// TwinCAT 3 PLC project RealFFT
// ProgramVersion: 3.1.4020.10
// libraries:
//   Tc2_Standard, * (Beckhoff Automation GmbH)
//   Tc2_System, * (Beckhoff Automation GmbH)
//   Tc2_Utilities, * (Beckhoff Automation GmbH)
//   Tc3_CM, * (Beckhoff Automation GmbH)
//   Tc3_CM_Base, * (Beckhoff Automation GmbH)
//   Tc3_Module, * (Beckhoff Automation GmbH)
//   Tc3_MultiArray, * (Beckhoff Automation GmbH)
// project tree:
//   DUTs/Error Monitoring/ ST_HRErrHist.TcDUT
//   DUTs/ E_AnalysisIDs.TcDUT
//   DUTs/Function Generator/ E_FunctionType.TcDUT
//   GVLs/ GVL_Constants.TcGVL
//   / PlcTask.TcTTO, PlcTaskCM.TcTTO
//   POUs/Error Monitoring/ FB_HRErrHist.TcPOU
//   POUs/Function Generator/ FB_FunctionGenerator.TcPOU
//   POUs/ MAIN.TcPOU, MAIN_CM.TcPOU
// real-time tasks:
//   TASK PlcTaskCM: cycle T#5ms, priority 6, ADS port 350
//   TASK PlcTask: cycle T#1ms, priority 4, ADS port 351

CONFIGURATION RealFFT
    RESOURCE PLC ON TwinCAT3
        TASK PlcTask(INTERVAL := T#1ms, PRIORITY := 4);
        TASK PlcTaskCM(INTERVAL := T#5ms, PRIORITY := 6);
        PROGRAM MAIN WITH PlcTask : MAIN;
        PROGRAM MAIN_CM WITH PlcTaskCM : MAIN_CM;
    END_RESOURCE
END_CONFIGURATION

// ---- DUTs/Error Monitoring/ST_HRErrHist.TcDUT
TYPE ST_HRErrHist :
STRUCT
{attribute 'displaymode':='hex'}
	hrErrCode	: HRESULT;
	sErrSource	: STRING(63);
	nErrCount	: UDINT;
END_STRUCT
END_TYPE

// ---- DUTs/E_AnalysisIDs.TcDUT
TYPE E_AnalysisIDs :
(
	(* analysis chain *)
	eID_Source := 1,
	eID_FFT,
	eID_Sink
	
) UDINT;
END_TYPE

// ---- DUTs/Function Generator/E_FunctionType.TcDUT
{attribute 'qualified_only'}
TYPE E_FunctionType :
(
	Sine,		// typical for vibrations originating from rotating machine
	Square,		// mixed sine signals good for analyzing spectrum
	Pulse,		// mixed sine signals good for analyzing spectrum
	Triangular,	// mixed sine signals good for analyzing spectrum
	Sawtooth,	// ramp-type vibrations, continuously increasing
	AM			// amplitude modulation: typical for vibrations originating from gear-tooth failure or bearing faults
);
END_TYPE

// ---- GVLs/GVL_Constants.TcGVL
VAR_GLOBAL CONSTANT
	
	cOversamples 	: UDINT 	:= 10;				 // number of oversamples
	cFFTLength		: UDINT		:= 2048;			 // length of FFT 
	cBufferLength	: UDINT		:= cFFTLength;	     // attention: needs to be equal to cFFTLength (no overlap)	
	cFFTResult 		: UDINT 	:= cFFTLength/2+1;	 // result of mag. spectrum - cFFTLength/2+1
		
END_VAR

// ---- POUs/MAIN.TcPOU
PROGRAM MAIN

VAR CONSTANT
    cInitSource			: ST_MA_MultiArray_InitPars 
							:= ( eTypeCode := eMA_TypeCode_LREAL, nDims := 1, aDimSizes := [cBufferLength]);	
END_VAR

VAR
	(* Input *)
	nInputSelection		: UDINT := 1;						// Switch between hardware and function generator	
	nSample				: UDINT;                            
	aEl3632 AT %I*		: ARRAY[1..cOversamples] OF INT;	// Input from hardware e.g. EL3632
	
	(* Signal Generator *)
	fbFunctionGenerator	: FB_FunctionGenerator;
	fSetFrequency		: LREAL := 200;		// Hz
	fSetAmplitude		: LREAL := 13;		// peak amplitude of sin signal, in Volts		
    fDC					: LREAL := 7;       // Amplitude of DC	
	
	(* Source buffers *)	
	aBuffer				: ARRAY[1..cOversamples] OF LREAL;				// local varibale -> to source				
	fbSource			: FB_CMA_Source :=(	stInitPars := cInitSource, 
											nOwnID := eID_Source, 
											aDestIDs := [eID_FFT]);		// Initialize source buffers
	(* Result buffers *)										
	aSpectrumResult		: ARRAY[1..cFFTResult] OF LCOMPLEX;				// local result variable <- from sink
    fbSink				: FB_CMA_Sink := (nOwnID := eID_Sink);			// Initialize sink buffers
	
	
	(* post-processing of fft *)
	nCountResults		: ULINT;							// increments for every fft calculation
	bCalculate			: BOOL;								// true if fft calculation ready	
	SpectrumAbs         : ARRAY[1..cFFTResult] OF LREAL; 	// magnitude spectrum variable 
	(* max amplitude calculation *)
	fMaxAmpl			: LREAL;
	nIdxOfMaxAmpl		: UDINT;							// index of max amplitude in spectrum result array 
	(* frequency calculation *)
	fSampleTaskCycleTime: LREAL := 1; // ms
	fSampleRate			: LREAL;      // Hz  ( sample rate = oversampling factor / cycle time )
	fResolution			: LREAL;      // Hz/Idx
	fFrequency			: LREAL;      // Hz	
	
	(* error monitoring *)
	fbErrHist			: FB_HRErrHist;

END_VAR

(* Input *) 
CASE nInputSelection OF
	0:  (* input from EL3632 *)
		FOR nSample := 1 TO cOversamples DO
			aBuffer[nSample] := INT_TO_LREAL(aEl3632[nSample]);
		END_FOR
	1:  (* signal generator *)		
		fbFunctionGenerator(	fFrequency 	:= fSetFrequency,
								fAmplitude 	:= fSetAmplitude,
								eFunction 	:= E_FunctionType.Sine,
								aSignal		:= aBuffer );		
        // add DC to signal
		FOR nSample := 1 TO cOversamples DO
			aBuffer[nSample] := fDC+aBuffer[nSample];
		END_FOR								
END_CASE					

(* Call source to collect data *)
fbSource.Input1D( pDataIn 			:= ADR(aBuffer),
				  nDataInSize 		:= SIZEOF(aBuffer), 
				  eElementType 		:= eMA_TypeCode_LREAL,
				  nWorkDim 			:= 0,
				  pStartIndex		:= 0,
				  nOptionPars		:= cCMA_Option_MarkInterruption ); 
IF fbSource.bError THEN
	fbErrHist.AddError(bErr:=TRUE, hrErrCode:=fbSource.hrErrorCode, sErrSource:='MAIN.fbSource'); // error monitoring
	// ToDo: if error
END_IF


(* Push results to sink *)
fbSink.Output1D(	pDataOut 		:= ADR(aSpectrumResult), 
					nDataOutSize 	:= SIZEOF(aSpectrumResult), 
					eElementType 	:= eMA_TypeCode_LCOMPLEX, 
					nWorkDim 		:= 0,
					nElements		:= 0,
					pStartIndex 	:= 0,
					nOptionPars		:= 0,
					bNewResult		=> bCalculate );
IF fbSink.bError THEN
	fbErrHist.AddError(bErr:=TRUE, hrErrCode:=fbSink.hrErrorCode, sErrSource:='MAIN.fbSink'); // error monitoring
	// ToDo: if error
END_IF

(* post-process fft result *)
IF bCalculate THEN
	nCountResults := fbSink.nCntResults;
	
	// Calculate absolute value as aSpectrumResult is of complex type
	FOR nSample := 1 TO cFFTResult DO			   	   
	   SpectrumAbs[nSample] := SQRT(aSpectrumResult[nSample].re * aSpectrumResult[nSample].re + aSpectrumResult[nSample].im * aSpectrumResult[nSample].im);
       
	   // scale spectrum
	   IF nSample = 1 THEN
		   SpectrumAbs[nSample] := SpectrumAbs[nSample]/cFFTLength;   // scale DC value
	   ELSE
		   SpectrumAbs[nSample] := 2*SpectrumAbs[nSample]/cFFTLength; // scale frequencies not equal to 0
	   END_IF
	   
	   
	END_FOR;
	
	IF NOT lrealisnan(SpectrumAbs[1]) THEN
		// Calculate max amplitude in spectrum
		fMaxAmpl := 0;
		FOR nSample:=1 TO cFFTResult DO
			IF SpectrumAbs[nSample] > fMaxAmpl THEN
				fMaxAmpl := SpectrumAbs[nSample];
				nIdxOfMaxAmpl := nSample;
			END_IF
		END_FOR
		
		// Calculate frequency for max amplitude [ frequency = index * (sample rate / FFT length) ]
		fSampleRate := cOversamples * (1000.0 / fSampleTaskCycleTime);
		fResolution := fSampleRate / cFFTLength;
		fFrequency := (nIdxOfMaxAmpl-1) * fResolution;	 // -1 to consider DC = 0*fResolution
	END_IF

	
END_IF

END_PROGRAM

// ---- POUs/Function Generator/FB_FunctionGenerator.TcPOU
// generates a signal build up by the specified function type. v1.6
FUNCTION_BLOCK FB_FunctionGenerator
VAR_INPUT
	bEnable		: BOOL 	:= TRUE;	// set TRUE to generate the specified signal; set FALSE to reset the signal buffer
	fFrequency	: LREAL := 1000;	// in [Hz]
	fAmplitude	: LREAL := 1;
	fOffset		: LREAL	:= 0;	
	nDutyCycle	: UINT 	:= 50;		// in [%] (for pulse function)
	eFunction	: E_FunctionType := E_FunctionType.Sine;	
END_VAR
VAR_IN_OUT
	aSignal		: ARRAY[1..cOversamples] OF LREAL;
END_VAR
VAR_OUTPUT
	bError		: BOOL;
END_VAR

VAR
	bInit						: BOOL := TRUE;
	fbGetTaskIdx				: GETCURTASKINDEX;
	
	fLastFrequency				: LREAL;		// in [Hz]
	fLastAmplitude				: LREAL;
	fLastOffset					: LREAL;
	nLastDutyCycle				: UINT;
	eLastFunction				: E_FunctionType;
	
	nSamples					: UDINT;
	fCycleTime					: LREAL;		// in [s]
	fDelta						: LREAL;		// amplitude delta per sample
	fPhase						: LREAL;		// in [°]
	nSign						: INT := 1;		// 1 or -1
	fLastSignalValue			: LREAL;		// amplitude
	fPeriod						: LREAL;		// in [s]
	fAngularIncrement			: LREAL;		// in [°]
	fAngularIncrementPerCycle	: LREAL;		// in [°]
	fAngularIncrementPerSample	: LREAL;		// in [°]
	(* for modulated signal (carrier signal without offset) *)
	fCarrierFrequency					: LREAL := 500;	// in [Hz] (sine)
	fCarrierAmplitude					: LREAL := 1;
	fCarrierPeriod						: LREAL;		// in [s]
	fCarrierAngularIncrement			: LREAL;		// in [°]
	fCarrierAngularIncrementPerCycle	: LREAL;		// in [°]
	fCarrierAngularIncrementPerSample	: LREAL;		// in [°]
				
END_VAR

IF bEnable THEN
	IF fLastFrequency <> fFrequency THEN
		bInit := TRUE; // For automatic initializing
		fLastFrequency := fFrequency;
	END_IF
	IF fLastAmplitude <> fAmplitude THEN
		bInit := TRUE; // For automatic initializing
		fLastAmplitude := fAmplitude;
	END_IF
	IF fLastOffset <> fOffset THEN
		bInit := TRUE; // For automatic initializing
		fLastOffset := fOffset;
	END_IF
	IF nLastDutyCycle <> nDutyCycle THEN
		bInit := TRUE; // For automatic initializing
		nLastDutyCycle := nDutyCycle;
	END_IF
	IF eLastFunction <> eFunction THEN
		bInit := TRUE; // For automatic initializing
		eLastFunction := eFunction;
	END_IF
	IF bInit THEN
		// Get task info	
		fbGetTaskIdx();
		fCycleTime := UDINT_TO_LREAL(TwinCAT_SystemInfoVarList._TaskInfo[fbGetTaskIdx.index].CycleTime) (*100ns*) / (10.0 * 1000.0 * 1000.0);	
		fLastSignalValue := 0;
		nSign := 1;
		fAngularIncrement := 0;
		// Flush out old data
		MEMSET(ADR(aSignal), 0, SIZEOF(aSignal));
		IF fFrequency > 0 AND fCycleTime > 0 THEN		
			// Calculate period, increments per plc cycle, increment per oversample
			IF cOversamples > 0 THEN			
				IF eFunction = E_FunctionType.Sine THEN
					fPeriod := 1/fFrequency;
					fAngularIncrementPerCycle := 360*(fCycleTime/fPeriod);
					fAngularIncrementPerSample := fAngularIncrementPerCycle/cOversamples;
					// no phase adjustment
					bInit := FALSE;	
				ELSIF eFunction = E_FunctionType.Square	THEN
					fPeriod := 1/fFrequency;
					fAngularIncrementPerCycle  := 360*(fCycleTime/fPeriod);
					fAngularIncrementPerSample := fAngularIncrementPerCycle/cOversamples;
					fPhase := 0.5*360;
					bInit := FALSE;
				ELSIF eFunction = E_FunctionType.Pulse THEN
					fPeriod := 1/fFrequency;
					fAngularIncrementPerCycle  := 360*(fCycleTime/fPeriod);
					fAngularIncrementPerSample := fAngularIncrementPerCycle/cOversamples;
					IF nDutyCycle > 100 THEN
						nDutyCycle := 100;
					END_IF
					fPhase := (UDINT_TO_LREAL(nDutyCycle)/100)*360;
					bInit := FALSE;					
				ELSIF eFunction = E_FunctionType.Triangular THEN
					fPeriod := 1/fFrequency;				
					fAngularIncrementPerCycle  := 360*(fCycleTime/fPeriod);
					fAngularIncrementPerSample := fAngularIncrementPerCycle/cOversamples;
					fPhase := 0.5*360; 
					fDelta := 4*(fAmplitude/(360/fAngularIncrementPerSample));				
					bInit := FALSE;
				ELSIF eFunction = E_FunctionType.Sawtooth THEN
					fPeriod := 1/fFrequency;			
					fAngularIncrementPerCycle  := 360*(fCycleTime/fPeriod);		
					fAngularIncrementPerSample := fAngularIncrementPerCycle/cOversamples;
					fDelta := fAmplitude/(360/fAngularIncrementPerSample);
					bInit := FALSE;
				ELSIF eFunction = E_FunctionType.AM THEN
					fPeriod := 1/fFrequency;
					fAngularIncrementPerCycle := 360*(fCycleTime/fPeriod);
					fAngularIncrementPerSample := fAngularIncrementPerCycle/cOversamples;
					// no phase adjustment
					fCarrierPeriod := 1/fCarrierFrequency;
					fCarrierAngularIncrementPerCycle := 360*(fCycleTime/fCarrierPeriod);
					fCarrierAngularIncrementPerSample := fCarrierAngularIncrementPerCycle/cOversamples;				
					// no phase adjustment	
					bInit := FALSE;
				ELSE
					bError := TRUE;	
				END_IF
			ELSE
				bError := TRUE;
			END_IF
		ELSE
			bError := TRUE;
		END_IF
	END_IF
	
	// Enable function generator
	IF NOT bError THEN		
		CASE eFunction OF		
			// sine: typical for vibrations originating from rotating machine
			E_FunctionType.Sine: Sine();
			
			// square: mixed sine signals good for analyzing spectrum				
			E_FunctionType.Square: Square();
			
			// pulse: mixed sine signals good for analyzing spectrum				
			E_FunctionType.Pulse: Pulse();
	
			// sawtooth: ramp-type vibrations, continuously increasing			
			E_FunctionType.Sawtooth: Sawtooth();
		
			// triangular: mixed sine signals good for analyzing spectrum
			E_FunctionType.Triangular: Triangular();
		
			// amplitude modulation: typical for vibrations originating from gear-tooth failure or bearing faults
			// Carrier signal with own frequency and amplitude		
			E_FunctionType.AM: AM();				
		END_CASE
	END_IF
ELSE
	// Flush out old data
	MEMSET(ADR(aSignal), 0, SIZEOF(aSignal));
	
	bInit := TRUE;
	bError := FALSE;
END_IF

METHOD PRIVATE AM
VAR_INPUT
END_VAR
{warning disable C0371}

FOR nSamples := 1 TO cOversamples DO
	// base signal * carrier signal
	aSignal[nSamples] := ( fAmplitude*SIN(2*PI*(fAngularIncrement+(nSamples-1)*fAngularIncrementPerSample)/360) + fOffset )
							* ( fCarrierAmplitude*SIN(2*PI*(fCarrierAngularIncrement+(nSamples-1)*fCarrierAngularIncrementPerSample)/360) );
END_FOR
// Increment angular positions
fAngularIncrement := fAngularIncrement + fAngularIncrementPerCycle;
fCarrierAngularIncrement := fCarrierAngularIncrement + fCarrierAngularIncrementPerCycle;

{warning restore C0371}
END_METHOD

METHOD PRIVATE Pulse
VAR_INPUT
END_VAR
{warning disable C0371}

FOR nSamples := 1 TO cOversamples DO
	// For pulse wave (unequal phases)
	IF (fAngularIncrement >= 360) THEN
		fAngularIncrement := fAngularIncrement - DINT_TO_LREAL(LREAL_TO_DINT(fAngularIncrement/360))*360;
		// or with Tc2_Math library: fAngularIncrement := LMOD(fAngularIncrement,360);
	END_IF
	IF (fAngularIncrement < fPhase) THEN
		nSign := 1;		
	ELSIF (fAngularIncrement >= fPhase) THEN
		nSign := 0;
	END_IF
	fAngularIncrement := fAngularIncrement + fAngularIncrementPerSample;
	
	aSignal[nSamples] := nSign*fAmplitude;
	
	aSignal[nSamples] := aSignal[nSamples] + fOffset;
END_FOR

{warning restore C0371}
END_METHOD

METHOD PRIVATE Sawtooth
VAR_INPUT
END_VAR
{warning disable C0371}

FOR nSamples := 1 TO cOversamples DO
	// For sawtooth wave (equal phase = period/2)
	IF (fAngularIncrement >= 360) THEN
		fAngularIncrement := fAngularIncrement - DINT_TO_LREAL(LREAL_TO_DINT(fAngularIncrement/360))*360;
		// or with Tc2_Math library: fAngularIncrement := LMOD(fAngularIncrement,360);
		fLastSignalValue := fLastSignalValue -fAmplitude;
	END_IF
	fAngularIncrement := fAngularIncrement + fAngularIncrementPerSample;

	aSignal[nSamples] := fLastSignalValue + fDelta;

	// Store last sample
	fLastSignalValue := aSignal[nSamples];
	
	aSignal[nSamples] := aSignal[nSamples] + fOffset;					
END_FOR	

{warning restore C0371}
END_METHOD

METHOD PRIVATE Sine
VAR_INPUT
END_VAR
{warning disable C0371}

FOR nSamples := 1 TO cOversamples DO
	aSignal[nSamples] := fAmplitude*SIN(2*PI*(fAngularIncrement+(nSamples-1)*fAngularIncrementPerSample)/360);

	aSignal[nSamples] := aSignal[nSamples] + fOffset;
END_FOR

// Increment angular position
fAngularIncrement := fAngularIncrement + fAngularIncrementPerCycle;

{warning restore C0371}
END_METHOD

METHOD PRIVATE Square
VAR_INPUT
END_VAR
{warning disable C0371}

FOR nSamples := 1 TO cOversamples DO
	// For square wave (equal phase = period/2)
	IF (fAngularIncrement >= 360) THEN
		fAngularIncrement := fAngularIncrement - DINT_TO_LREAL(LREAL_TO_DINT(fAngularIncrement/360))*360;
		// or with Tc2_Math library: fAngularIncrement := LMOD(fAngularIncrement,360);
	END_IF
	IF (fAngularIncrement < fPhase) THEN
		nSign := 1;
	ELSIF (fAngularIncrement >= fPhase) THEN
		nSign := -1;
	END_IF
	fAngularIncrement := fAngularIncrement + fAngularIncrementPerSample;
	
	aSignal[nSamples] := nSign*fAmplitude;
	
	aSignal[nSamples] := aSignal[nSamples] + fOffset;
END_FOR

{warning restore C0371}
END_METHOD

METHOD PRIVATE Triangular
VAR_INPUT
END_VAR
{warning disable C0371}

FOR nSamples := 1 TO cOversamples DO
	IF (fAngularIncrement >= 360) THEN
		fAngularIncrement := fAngularIncrement - DINT_TO_LREAL(LREAL_TO_DINT(fAngularIncrement/360))*360;
		// or with Tc2_Math library: fAngularIncrement := LMOD(fAngularIncrement,360);
	END_IF
	// Negative delta -> Positive delta
	IF fAngularIncrement < fPhase/2 THEN	
		nSign := 1;		
	ELSIF fAngularIncrement >= fPhase/2 AND fAngularIncrement < 3*fPhase/2 THEN
		nSign := -1;
	ELSIF fAngularIncrement >= 3*fPhase/2 THEN
		nSign := 1;	
	END_IF
	fAngularIncrement := fAngularIncrement + fAngularIncrementPerSample;
	
	aSignal[nSamples] := fLastSignalValue + nSign*fDelta;
	IF aSignal[nSamples] > fAmplitude THEN
		aSignal[nSamples] := aSignal[nSamples] - 2*(aSignal[nSamples]-fAmplitude);
	ELSIF aSignal[nSamples] < (-1)*fAmplitude THEN
		aSignal[nSamples] := aSignal[nSamples] - 2*(aSignal[nSamples]+fAmplitude);
	END_IF
	
	// Store last sample
	fLastSignalValue := aSignal[nSamples];		
	
	aSignal[nSamples] := aSignal[nSamples] + fOffset;
END_FOR

{warning restore C0371}
END_METHOD

END_FUNCTION_BLOCK

// ---- POUs/Error Monitoring/FB_HRErrHist.TcPOU
FUNCTION_BLOCK FB_HRErrHist
(* v1.10
build up an error history consisting of two arrays and one index.
The index shows the actual array position. The last error id and the count for this id are saved in the arrays.
If an error id is the same as the previous input error the counter is increased. Otherwise the index is increased.
*)
VAR_INPUT
	bEdgeDetect	: BOOL;	(* FALSE: every input(bErr) is processed; TRUE: only rising edge of input is processed *)
END_VAR
VAR_OUTPUT
	nErrSum		: UINT;
	nErrIdx		: UINT; // error list index of last occured error (max. cHistLen)
	aErrList	: ARRAY[1..cHistLen] OF ST_HRErrHist;
END_VAR

VAR
	bNewErr		: BOOL;
	fbErrTrig	: R_TRIG;
END_VAR
VAR CONSTANT
	cHistLen	: UINT := 100;
END_VAR

METHOD AddError
VAR_INPUT
	bErr		: BOOL;
	hrErrCode	: HRESULT;
	sErrSource	: STRING(63);
END_VAR
fbErrTrig(CLK:=bErr);
IF bEdgeDetect THEN
	bNewErr := fbErrTrig.Q;
ELSE
	bNewErr := bErr;
END_IF

IF bNewErr THEN
	nErrSum := nErrSum + 1;
	IF nErrIdx < cHistLen THEN
		IF nErrIdx = 0 THEN
			nErrIdx	:= nErrIdx + 1;
		ELSIF aErrList[nErrIdx].hrErrCode <> hrErrCode OR aErrList[nErrIdx].sErrSource <> sErrSource THEN
			nErrIdx	:= nErrIdx + 1;
		END_IF
		aErrList[nErrIdx].hrErrCode := hrErrCode;
		aErrList[nErrIdx].sErrSource := sErrSource;
		aErrList[nErrIdx].nErrCount := aErrList[nErrIdx].nErrCount + 1;
	END_IF
END_IF
END_METHOD

METHOD Reset
VAR_INPUT
END_VAR
nErrSum := 0;
nErrIdx := 0;
MEMSET(ADR(aErrList),0,SIZEOF(aErrList));
END_METHOD

END_FUNCTION_BLOCK

// ---- POUs/MAIN_CM.TcPOU
PROGRAM MAIN_CM
VAR CONSTANT										
	cInitFFT 	: ST_CM_RealFFT_InitPars := (	nFFT_Length := cFFTLength, bForward := TRUE);															
END_VAR

VAR													
	fbRealFFT			: FB_CMA_RealFFT :=(	stInitPars := cInitFFT, nOwnID := eID_FFT, aDestIDs := [eID_Sink] );														
	fbErrHist			: FB_HRErrHist; // error monitoring
END_VAR


// Call RealFFT 
fbRealFFT.Call();
IF fbRealFFT.bError THEN
	fbErrHist.AddError(bErr:=TRUE, hrErrCode:=fbRealFFT.hrErrorCode, sErrSource:='MAIN_CM.fbRealFFT'); // error monitoring
	// ToDo: if error
END_IF

END_PROGRAM
